PROGRAM lightComboErrorChecks
VAR
END_VAR
VAR // added by the converter: edge detectors and wires of the graphical bodies
    _w1, _w2, _w3, _w4, _w5, _w6, _w7, _w8 : BOOL;
END_VAR

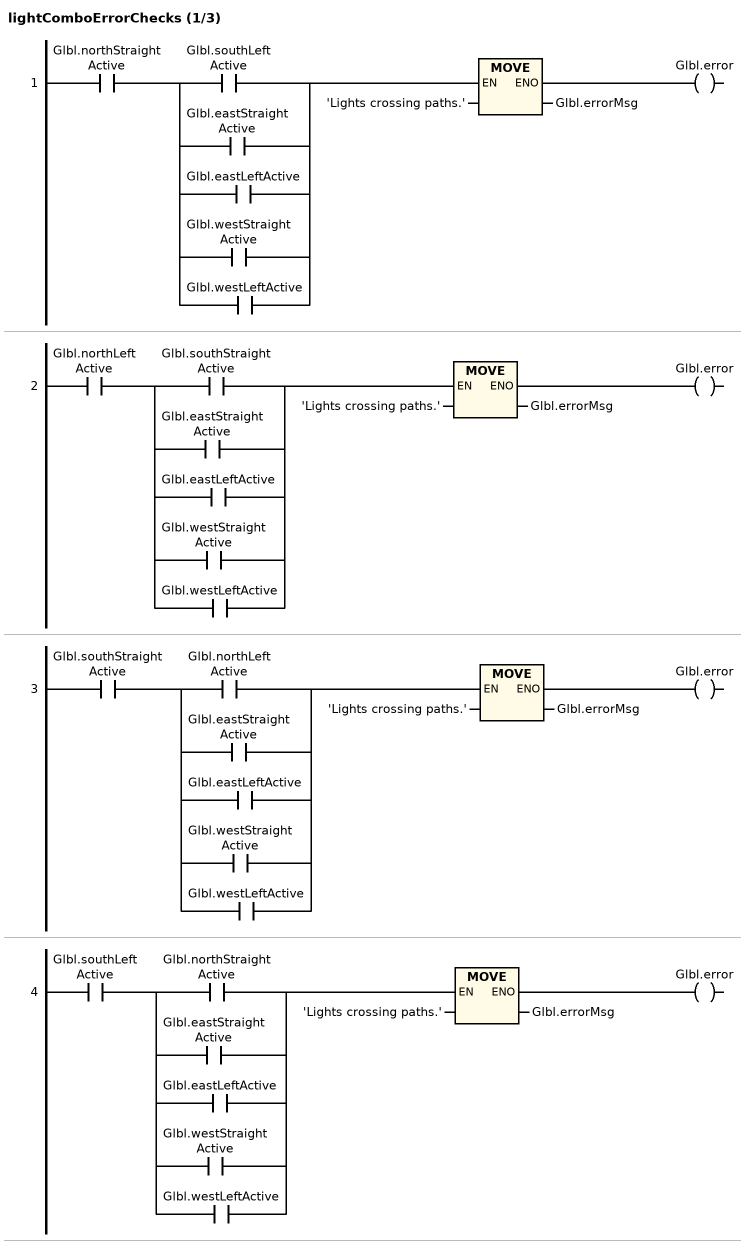
// NETWORK 1
_w1 := Glbl.northStraightActive AND (Glbl.southLeftActive OR Glbl.eastStraightActive OR Glbl.eastLeftActive OR Glbl.westStraightActive OR Glbl.westLeftActive);
IF _w1 THEN Glbl.errorMsg := 'Lights crossing paths.'; END_IF
Glbl.error := _w1;

// NETWORK 2
_w2 := Glbl.northLeftActive AND (Glbl.southStraightActive OR Glbl.eastStraightActive OR Glbl.eastLeftActive OR Glbl.westStraightActive OR Glbl.westLeftActive);
IF _w2 THEN Glbl.errorMsg := 'Lights crossing paths.'; END_IF
Glbl.error := _w2;

// NETWORK 3
_w3 := Glbl.southStraightActive AND (Glbl.northLeftActive OR Glbl.eastStraightActive OR Glbl.eastLeftActive OR Glbl.westStraightActive OR Glbl.westLeftActive);
IF _w3 THEN Glbl.errorMsg := 'Lights crossing paths.'; END_IF
Glbl.error := _w3;

// NETWORK 4
_w4 := Glbl.southLeftActive AND (Glbl.northStraightActive OR Glbl.eastStraightActive OR Glbl.eastLeftActive OR Glbl.westStraightActive OR Glbl.westLeftActive);
IF _w4 THEN Glbl.errorMsg := 'Lights crossing paths.'; END_IF
Glbl.error := _w4;

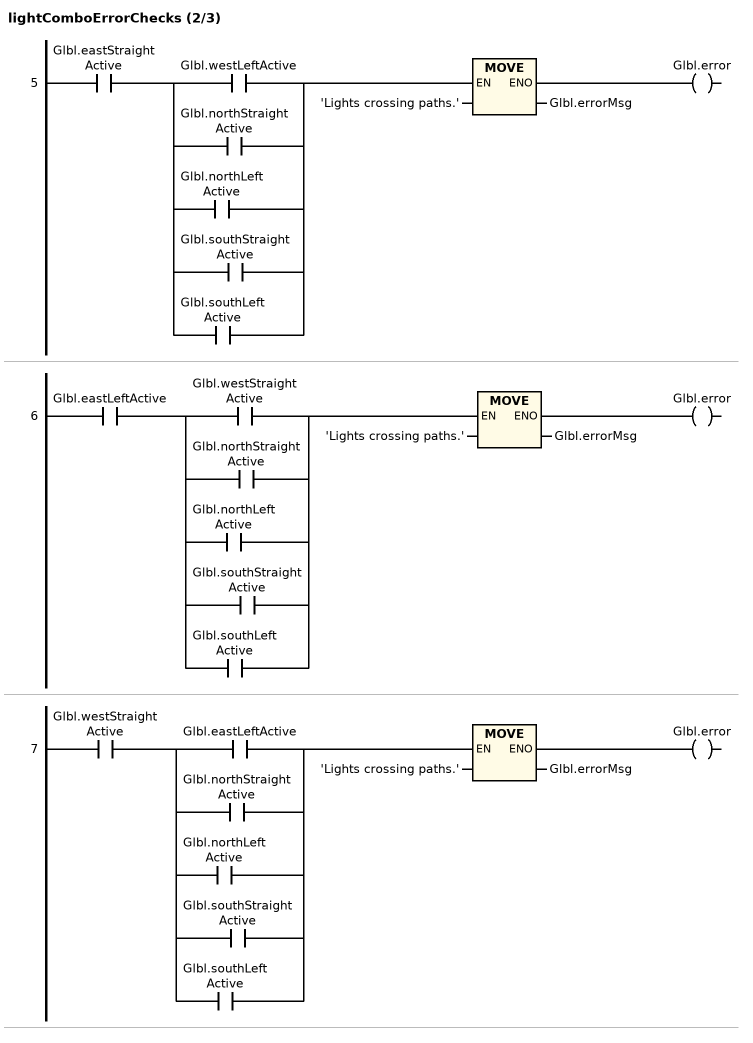
// NETWORK 5
_w5 := Glbl.eastStraightActive AND (Glbl.westLeftActive OR Glbl.northStraightActive OR Glbl.northLeftActive OR Glbl.southStraightActive OR Glbl.southLeftActive);
IF _w5 THEN Glbl.errorMsg := 'Lights crossing paths.'; END_IF
Glbl.error := _w5;

// NETWORK 6
_w6 := Glbl.eastLeftActive AND (Glbl.westStraightActive OR Glbl.northStraightActive OR Glbl.northLeftActive OR Glbl.southStraightActive OR Glbl.southLeftActive);
IF _w6 THEN Glbl.errorMsg := 'Lights crossing paths.'; END_IF
Glbl.error := _w6;

// NETWORK 7
_w7 := Glbl.westStraightActive AND (Glbl.eastLeftActive OR Glbl.northStraightActive OR Glbl.northLeftActive OR Glbl.southStraightActive OR Glbl.southLeftActive);
IF _w7 THEN Glbl.errorMsg := 'Lights crossing paths.'; END_IF
Glbl.error := _w7;

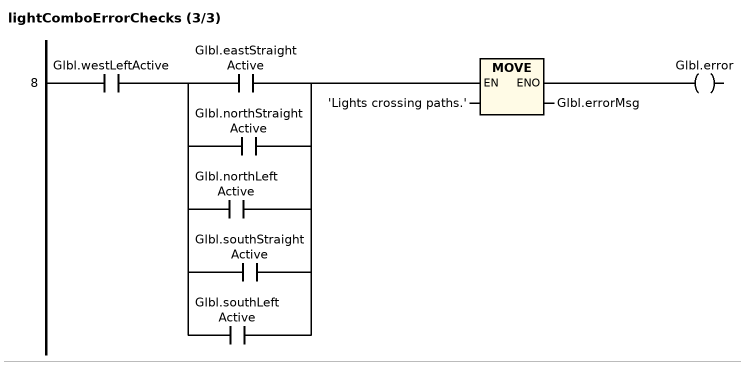
// NETWORK 8
_w8 := Glbl.westLeftActive AND (Glbl.eastStraightActive OR Glbl.northStraightActive OR Glbl.northLeftActive OR Glbl.southStraightActive OR Glbl.southLeftActive);
IF _w8 THEN Glbl.errorMsg := 'Lights crossing paths.'; END_IF
Glbl.error := _w8;

END_PROGRAM

(* stored: Version 1.1.0.1, ProductVersion 3.1.4022.10
   POU lightComboErrorChecks: Id {15cf21ee-d398-48b0-81f1-e34bdd9f6040}, SpecialFunc None *)
